// Mitsubishi GX Works2 project: 실행 프로그램 나누기   PLC: Q03UDV

PROGRAM MAIN
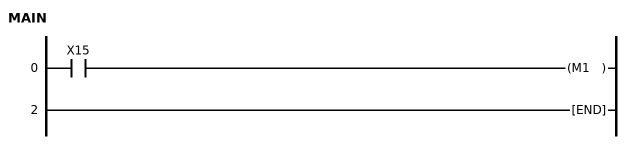
0     LD      X15
      OUT     M1
2     END
END_PROGRAM

PROGRAM OUTPUT
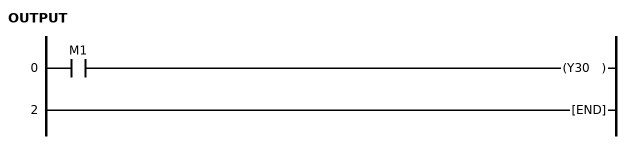
0     LD      M1
      OUT     Y30
2     END
END_PROGRAM
